KUKA KRL program: home2wait.src, home2wait.dat

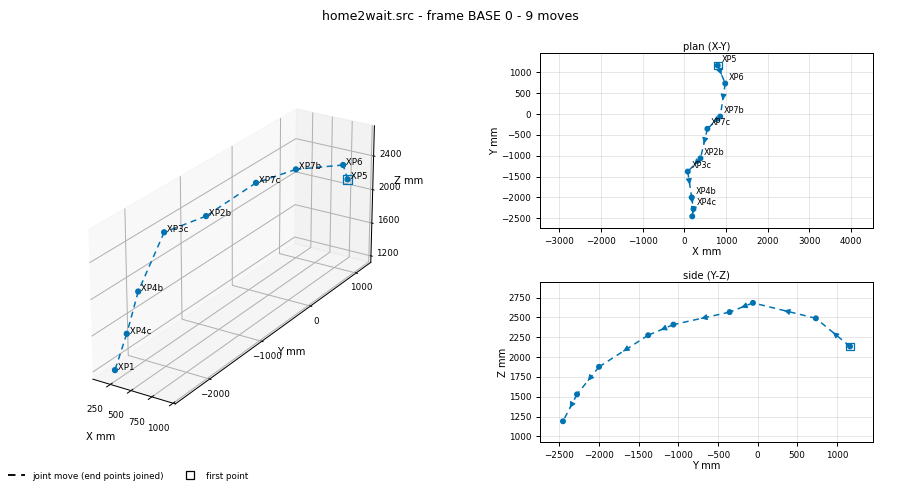
[picture p0: tool path of home2wait.src in frame BASE 0, 9 of 11 moves have a stored position in this frame; points joined in program order, loops and branches not executed]
--- home2wait.src ---
&ACCESS RVO1
&REL 27
&PARAM TEMPLATE = C:\KRC\Roboter\Template\vorgabe
&PARAM EDITMASK = *
DEF home2wait( )

;================================================
; MODELO   : C-520
; IE GRUPO : 5J
; ESTACION : 85
; ROBOT    : 85r01
; FUNCION  : xxxxxxx
;================================================

;FOLD INI
  ;FOLD BASISTECH INI
    GLOBAL INTERRUPT DECL 3 WHEN $STOPMESS==TRUE DO IR_STOPM ( )
    INTERRUPT ON 3
    BAS (#INITMOV,0 )
  ;ENDFOLD (BASISTECH INI)
;FOLD SPOTTECH INI
;USERSPOT(#INIT)
;ENDFOLD (SPOTTECH INI)
;FOLD GRIPPERTECH INI
USER_GRP(0,DUMMY,DUMMY,GDEFAULT)
INTERRUPT DECL 20 WHEN $FLAG[20]==FALSE DO GRPS(#MON_ERR,20)
;ENDFOLD (GRIPPERTECH INI)
  ;FOLD USER INI
    ;Make your modifications here

  ;ENDFOLD (USER INI)
;ENDFOLD (INI)

;FOLD PTP HOME CONT Vel=100 % DEFAULT;%{PE}%R 5.6.13,%MKUKATPBASIS,%CMOVE,%VPTP,%P 1:PTP, 2:HOME, 3:C_PTP, 5:100, 7:DEFAULT
$BWDSTART=FALSE
PDAT_ACT=PDEFAULT
FDAT_ACT=FHOME
BAS(#PTP_PARAMS,100)
$H_POS=XHOME
PTP XHOME C_PTP
;ENDFOLD

;FOLD PTP P5 CONT Vel=100 % H Tool[12] Base[0];%{PE}%R 5.6.13,%MKUKATPBASIS,%CMOVE,%VPTP,%P 1:PTP, 2:P5, 3:C_PTP, 5:100, 7:H
$BWDSTART=FALSE
PDAT_ACT=PH
FDAT_ACT=FP5
BAS(#PTP_PARAMS,100)
PTP XP5 C_PTP
;ENDFOLD

;ENTRAR_DEDOS()
;FOLD OUT 88 'toPLC waiting sensor' State=TRUE CONT;%{PE}%R 5.6.13,%MKUKATPBASIS,%COUT,%VOUTX,%P 2:88, 3:toPLC waiting sensor, 5:TRUE, 6:CONTINUE
CONTINUE
$OUT[88]=TRUE
;ENDFOLD
;FOLD OUT 97 'dedos fuera' State=FALSE CONT;%{PE}%R 5.6.13,%MKUKATPBASIS,%COUT,%VOUTX,%P 2:97, 3:dedos fuera, 5:FALSE, 6:CONTINUE
CONTINUE
$OUT[97]=FALSE
;ENDFOLD
;FOLD OUT 98 'dedos dentro' State=TRUE CONT;%{PE}%R 5.6.13,%MKUKATPBASIS,%COUT,%VOUTX,%P 2:98, 3:dedos dentro, 5:TRUE, 6:CONTINUE
CONTINUE
$OUT[98]=TRUE
;ENDFOLD

;FOLD PTP P6 CONT Vel=100 % M Tool[12] Base[0];%{PE}%R 5.6.13,%MKUKATPBASIS,%CMOVE,%VPTP,%P 1:PTP, 2:P6, 3:C_PTP, 5:100, 7:M
$BWDSTART=FALSE
PDAT_ACT=PM
FDAT_ACT=FP6
BAS(#PTP_PARAMS,100)
PTP XP6 C_PTP
;ENDFOLD
;FOLD PTP P7b CONT Vel=100 % M Tool[12] Base[0];%{PE}%R 5.6.13,%MKUKATPBASIS,%CMOVE,%VPTP,%P 1:PTP, 2:P7b, 3:C_PTP, 5:100, 7:M
$BWDSTART=FALSE
PDAT_ACT=PM
FDAT_ACT=FP7b
BAS(#PTP_PARAMS,100)
PTP XP7b C_PTP
;ENDFOLD

;FOLD WAIT FOR ( NOT IN 65 '201S161A dedos fuera izq' AND IN 66 '201S161B dedos dentro izq' AND NOT IN 97 '201S162A dedos fuera drch' AND IN 98 '201S162B dedos atras drch' ) CONT;%{PE}%R 5.6.13,%MKUKATPBASIS,%CEXT_WAIT_FOR,%VEXT_WAIT_FOR,%P 2:, 4:NOT, 5:$IN, 6:65, 7:201S161A dedos fuera izq, 8:AND, 9:, 10:$IN, 11:66, 12:201S161B dedos dentro izq, 13:AND, 14:NOT, 15:$IN, 16:97, 17:201S162A dedos fuera drch, 18:AND, 19:, 20:$IN, 21:98, 22:201S162B dedos atras drch, 24:CONTINUE
CONTINUE
WAIT FOR  (  NOT $IN[65] AND $IN[66] AND  NOT $IN[97] AND $IN[98] )
;ENDFOLD
;FOLD OUT 88 'toPLC waiting sensor' State=FALSE CONT;%{PE}%R 5.6.13,%MKUKATPBASIS,%COUT,%VOUTX,%P 2:88, 3:toPLC waiting sensor, 5:FALSE, 6:CONTINUE
CONTINUE
$OUT[88]=FALSE
;ENDFOLD

;FOLD PTP P7c CONT Vel=100 % H Tool[12] Base[0];%{PE}%R 5.6.13,%MKUKATPBASIS,%CMOVE,%VPTP,%P 1:PTP, 2:P7c, 3:C_PTP, 5:100, 7:H
$BWDSTART=FALSE
PDAT_ACT=PH
FDAT_ACT=FP7c
BAS(#PTP_PARAMS,100)
PTP XP7c C_PTP
;ENDFOLD
;FOLD PTP P2b CONT Vel=100 % H Tool[12] Base[0];%{PE}%R 5.6.13,%MKUKATPBASIS,%CMOVE,%VPTP,%P 1:PTP, 2:P2b, 3:C_PTP, 5:100, 7:H
$BWDSTART=FALSE
PDAT_ACT=PH
FDAT_ACT=FP2b
BAS(#PTP_PARAMS,100)
PTP XP2b C_PTP
;ENDFOLD
;FOLD PTP P3c CONT Vel=100 % H Tool[12] Base[0];%{PE}%R 5.6.13,%MKUKATPBASIS,%CMOVE,%VPTP,%P 1:PTP, 2:P3c, 3:C_PTP, 5:100, 7:H
$BWDSTART=FALSE
PDAT_ACT=PH
FDAT_ACT=FP3c
BAS(#PTP_PARAMS,100)
PTP XP3c C_PTP
;ENDFOLD
;FOLD PTP P4b CONT Vel=100 % H Tool[12] Base[0];%{PE}%R 5.6.13,%MKUKATPBASIS,%CMOVE,%VPTP,%P 1:PTP, 2:P4b, 3:C_PTP, 5:100, 7:H
$BWDSTART=FALSE
PDAT_ACT=PH
FDAT_ACT=FP4b
BAS(#PTP_PARAMS,100)
PTP XP4b C_PTP
;ENDFOLD
;FOLD PTP P4c CONT Vel=100 % H Tool[12] Base[0];%{PE}%R 5.6.13,%MKUKATPBASIS,%CMOVE,%VPTP,%P 1:PTP, 2:P4c, 3:C_PTP, 5:100, 7:H
$BWDSTART=FALSE
PDAT_ACT=PH
FDAT_ACT=FP4c
BAS(#PTP_PARAMS,100)
PTP XP4c C_PTP
;ENDFOLD
;FOLD PTP P1 CONT Vel=100 % H Tool[12] Base[0];%{PE}%R 5.6.13,%MKUKATPBASIS,%CMOVE,%VPTP,%P 1:PTP, 2:P1, 3:C_PTP, 5:100, 7:H
$BWDSTART=FALSE
PDAT_ACT=PH
FDAT_ACT=FP1
BAS(#PTP_PARAMS,100)
PTP XP1 C_PTP
;ENDFOLD

ENTRAR_DEDOS()
CERRAR_DEDOS()
ENTRAR_RODILLO()
ABRIR_CILINDRO_IP()
CLAMPAR_GONDOLA()

;FOLD PTP P8 Vel=100 % H Tool[14]:camara Base[19]:carrusel bien;%{PE}%R 5.6.13,%MKUKATPBASIS,%CMOVE,%VPTP,%P 1:PTP, 2:P8, 3:, 5:100, 7:H
$BWDSTART=FALSE
PDAT_ACT=PH
FDAT_ACT=FP8
BAS(#PTP_PARAMS,100)
PTP XP8
;ENDFOLD

;FOLD FORDTECH.Area_Req 1 Safety Position, 0 Return To Home, 1;%{PE}%MKUKATPUSER
Area_Req (1,0,1)
IF I_RETHP then
;goto home
ENDIF
;ENDFOLD

END

--- home2wait.dat ---
&ACCESS RVO1
&REL 27
&PARAM TEMPLATE = C:\KRC\Roboter\Template\vorgabe
&PARAM EDITMASK = *
DEFDAT  HOME2WAIT
;FOLD EXTERNAL DECLARATIONS;%{PE}%MKUKATPBASIS,%CEXT,%VCOMMON,%P
;FOLD GRIPPERTECH EXT
EXT  H50 (INT  :IN,INT  :IN,INT  :IN,GRP_TYP  :IN )
;ENDFOLD (GRIPPERTECH EXT)
;FOLD SPOTTECH EXT
EXT  USERSPOT (S_COMMAND  :IN,SPOT_TYPE  :IN )
;ENDFOLD (SPOTTECH EXT)
;FOLD BASISTECH EXT;%{PE}%MKUKATPBASIS,%CEXT,%VEXT,%P
EXT  BAS (BAS_COMMAND  :IN,REAL  :IN )
DECL INT SUCCESS
;ENDFOLD (BASISTECH EXT)
;FOLD USER EXT;%{E}%MKUKATPUSER,%CEXT,%VEXT,%P
;Make here your modifications

;ENDFOLD (USER EXT)
;ENDFOLD (EXTERNAL DECLARATIONS)
DECL BASIS_SUGG_T LAST_BASIS={POINT1[] "P7c                     ",POINT2[] "P7c                     ",CP_PARAMS[] "CPDAT0                  ",PTP_PARAMS[] "H                       ",CONT[] "C_PTP                   ",CP_VEL[] "2.0                     ",PTP_VEL[] "100                     ",SYNC_PARAMS[] "SYNCDAT                 ",SPL_NAME[] "S0                      "}
DECL PDAT PPDAT0={VEL 100.0,ACC 100.0,APO_DIST 100.0}
DECL E6POS XP0={X 2993.78296,Y -282.495789,Z 1156.71399,A -162.6474,B -2.34018302,C -91.4635925,S 2,T 43,E1 0.0,E2 0.0,E3 0.0,E4 0.0,E5 0.0,E6 0.0}
DECL FDAT FP0={TOOL_NO 3,BASE_NO 0,IPO_FRAME #BASE,POINT2[] " ",TQ_STATE FALSE}
DECL E6POS XP1={X 189.885101,Y -2452.52393,Z 1190.57898,A -179.364105,B 44.0344391,C 178.150208,S 2,T 10,E1 0.0,E2 0.0,E3 0.0,E4 0.0,E5 0.0,E6 0.0}
DECL FDAT FP1={TOOL_NO 12,BASE_NO 0,IPO_FRAME #BASE,POINT2[] " ",TQ_STATE FALSE}
DECL PDAT PPDAT1={VEL 100.0,ACC 100.0,APO_DIST 100.0,APO_MODE #CPTP}
DECL PDAT PPDAT2={VEL 100.0,ACC 100.0,APO_DIST 100.0,APO_MODE #CPTP}
DECL E6POS XP2={X 589.351379,Y -468.337097,Z 2436.07593,A -157.786194,B 16.6084003,C -176.289505,S 2,T 10,E1 0.0,E2 0.0,E3 0.0,E4 0.0,E5 0.0,E6 0.0}
DECL FDAT FP2={TOOL_NO 12,BASE_NO 0,IPO_FRAME #BASE,POINT2[] " ",TQ_STATE FALSE}
DECL PDAT PPDAT3={VEL 100.0,ACC 100.0,APO_DIST 100.0}
DECL E6POS XP3={X 670.961914,Y -761.631775,Z 2263.86011,A -169.724503,B 10.7614298,C 171.791306,S 2,T 10,E1 0.0,E2 0.0,E3 0.0,E4 0.0,E5 0.0,E6 0.0}
DECL FDAT FP3={TOOL_NO 0,BASE_NO 0,IPO_FRAME #BASE,POINT2[] " ",TQ_STATE FALSE}
DECL PDAT PPDAT4={VEL 100.0,ACC 100.0,APO_DIST 100.0,APO_MODE #CPTP}
DECL E6POS XP4={X 393.983398,Y -2048.18188,Z 1790.35803,A -175.634598,B 35.368969,C 177.474197,S 2,T 10,E1 0.0,E2 0.0,E3 0.0,E4 0.0,E5 0.0,E6 0.0}
DECL FDAT FP4={TOOL_NO 12,BASE_NO 0,IPO_FRAME #BASE,POINT2[] " ",TQ_STATE FALSE}
DECL PDAT PPDAT5={VEL 100.0,ACC 100.0,APO_DIST 100.0,APO_MODE #CPTP}
DECL E6POS XP5={X 801.582214,Y 1166.55701,Z 2133.69409,A -36.2449303,B 64.0939331,C -137.098602,S 2,T 11,E1 0.0,E2 0.0,E3 0.0,E4 0.0,E5 0.0,E6 0.0}
DECL FDAT FP5={TOOL_NO 12,BASE_NO 0,IPO_FRAME #BASE,POINT2[] " ",TQ_STATE FALSE}
DECL PDAT PPDAT6={VEL 100.0,ACC 100.0,APO_DIST 100.0,APO_MODE #CPTP}
DECL E6POS XP6={X 981.518372,Y 735.967224,Z 2488.48901,A -60.3836784,B 46.7860603,C -152.051498,S 2,T 11,E1 0.0,E2 0.0,E3 0.0,E4 0.0,E5 0.0,E6 0.0}
DECL FDAT FP6={TOOL_NO 12,BASE_NO 0,IPO_FRAME #BASE,POINT2[] " ",TQ_STATE FALSE}
DECL PDAT PPDAT7={VEL 100.0,ACC 100.0,APO_DIST 100.0,APO_MODE #CPTP}
DECL E6POS XP7={X 951.687195,Y 98.2863235,Z 2527.25293,A -116.173302,B 17.4556007,C -176.554199,S 2,T 11,E1 0.0,E2 0.0,E3 0.0,E4 0.0,E5 0.0,E6 0.0}
DECL FDAT FP7={TOOL_NO 12,BASE_NO 0,IPO_FRAME #BASE,POINT2[] " ",TQ_STATE FALSE}
DECL E6POS XP8={X -107.759399,Y -9.55283928,Z -929.549011,A 89.7361603,B 0.775884986,C 0.201503307,S 2,T 10,E1 0.0,E2 0.0,E3 0.0,E4 0.0,E5 0.0,E6 0.0}
DECL FDAT FP8={TOOL_NO 14,BASE_NO 19,IPO_FRAME #BASE,POINT2[] " ",TQ_STATE FALSE}
DECL PDAT PPDAT8={VEL 100.0,ACC 100.0,APO_DIST 100.0}
DECL PDAT PH={VEL 100.0,ACC 100.0,APO_DIST 100.0,APO_MODE #CPTP}
DECL E6POS XP100={X 224.123901,Y -2191.58203,Z 1632.96204,A -176.286499,B 38.0749092,C 177.541901,S 2,T 10,E1 0.0,E2 0.0,E3 0.0,E4 0.0,E5 0.0,E6 0.0}
DECL FDAT FP100={TOOL_NO 12,BASE_NO 0,IPO_FRAME #BASE,POINT2[] " ",TQ_STATE FALSE}
DECL E6POS XP4b={X 176.394302,Y -1997.90601,Z 1876.83704,A 171.723602,B 38.475029,C 175.432999,S 2,T 10,E1 0.0,E2 0.0,E3 0.0,E4 0.0,E5 0.0,E6 0.0}
DECL FDAT FP4b={TOOL_NO 12,BASE_NO 0,IPO_FRAME #BASE,POINT2[] " ",TQ_STATE FALSE}
DECL E6POS XP2B={X 387.577789,Y -1060.224,Z 2409.31494,A 175.079407,B 28.2810097,C 176.8965,S 2,T 10,E1 0.0,E2 0.0,E3 0.0,E4 0.0,E5 0.0,E6 0.0}
DECL FDAT FP2b={TOOL_NO 12,BASE_NO 0,IPO_FRAME #BASE,POINT2[] " ",TQ_STATE FALSE}
DECL E6POS XP3B={X 756.340881,Y -1237.66699,Z 2259.48096,A -167.671494,B 23.8709106,C 176.691299,S 2,T 10,E1 0.0,E2 0.0,E3 0.0,E4 0.0,E5 0.0,E6 0.0}
DECL FDAT FP3b={TOOL_NO 12,BASE_NO 0,IPO_FRAME #BASE,POINT2[] " ",TQ_STATE FALSE}
DECL E6POS XP3C={X 81.989502,Y -1378.06006,Z 2275.33496,A 163.519608,B 32.630661,C 173.996002,S 2,T 10,E1 0.0,E2 0.0,E3 0.0,E4 0.0,E5 0.0,E6 0.0}
DECL FDAT FP3c={TOOL_NO 12,BASE_NO 0,IPO_FRAME #BASE,POINT2[] " ",TQ_STATE FALSE}
DECL E6POS XP4C={X 219.222397,Y -2275.33203,Z 1530.021,A 177.485596,B 41.6465187,C 175.996002,S 2,T 10,E1 0.0,E2 0.0,E3 0.0,E4 0.0,E5 0.0,E6 0.0}
DECL FDAT FP4c={TOOL_NO 12,BASE_NO 0,IPO_FRAME #BASE,POINT2[] " ",TQ_STATE FALSE}
DECL E6POS XP7B={X 860.85498,Y -57.175499,Z 2683.31689,A -144.020004,B 36.9467392,C -174.620895,S 2,T 10,E1 0.0,E2 0.0,E3 0.0,E4 0.0,E5 0.0,E6 0.0}
DECL FDAT FP7b={TOOL_NO 12,BASE_NO 0,IPO_FRAME #BASE,POINT2[] " ",TQ_STATE FALSE}
DECL E6POS XP7C={X 552.763977,Y -351.462097,Z 2566.83398,A -166.712601,B 25.0852795,C -176.615295,S 2,T 10,E1 0.0,E2 0.0,E3 0.0,E4 0.0,E5 0.0,E6 0.0}
DECL FDAT FP7c={TOOL_NO 12,BASE_NO 0,IPO_FRAME #BASE,POINT2[] " ",TQ_STATE FALSE}
DECL PDAT PM={VEL 100.0,ACC 50.0,APO_DIST 100.0,APO_MODE #CPTP}
DECL PDAT PL={VEL 100.0,ACC 50.0,APO_DIST 100.0,APO_MODE #CPTP}
ENDDAT
